PROGRAM PRG_ControllerMode

VAR
	fbControllerMode : FB_ControllerMode;
END_VAR

// Runs FB with given values
fbControllerMode(
	bAuto := G_Inputs.bAuto, 			// Auto mode controller
	bManual := G_Inputs.bManual, 		// Manual mode controller
	bStart := G_Inputs.bStartButton,	// Start button
	bStop := G_Inputs.bStopButton, 		// Stop button
	
	// Values from FB sent to GVL
	bRunning => G_Mode.bRunning,		// System running
	bRunning => G_Output.bRunning,		// System running
	bManualMode => G_Mode.bManual,		// Manual mode
	bAutoMode => G_Mode.bAuto			// Auto mode
);

END_PROGRAM

(* stored: Version 1.1.0.1
   POU PRG_ControllerMode: Id {0450d79d-8ebf-4b0d-8196-6efb5a4dcb4c}, SpecialFunc None *)
